TYPE Tank_Ctx :
STRUCT
	io		: Tank_Io;
	hmi		: Tank_Hmi;
	priv	: Tank_Priv;
	state	: Tank_States;
END_STRUCT
END_TYPE

(* stored: Version 1.1.0.1
   DUT Tank_Ctx: Id {36b20bb0-ce77-4c98-acf0-fba43b62b034} *)
